PROGRAM P_PersistentDataSave
VAR
	fbSaveChanges :FB_Save;
	sFolderPath: STRING(255) := 'C:\Recipe_changes\';
END_VAR

IF P_persistent.bWritePersistent THEN
	fbSaveChanges.sFilePath := CONCAT(sFolderPath, 'Recipe_change');
    fbSaveChanges.sFilePath := CONCAT(fbSaveChanges.sFilePath, p_24h_C1_2.sCurrentDate);
    fbSaveChanges.sFilePath := CONCAT(fbSaveChanges.sFilePath, '.csv');
	fbSaveChanges();
END_IF

END_PROGRAM

(* stored: Version 1.1.0.1, ProductVersion 3.1.4026.13, FileIdentifier 561e912806da75a3470abee4b195e8b78ff5e6da, FileSignature 91b75a5166293d134c0b4d7ecb5ce9b6fdae071e385e36b36b597e2cd0a9c5db319be4bb0085fbdef6d3f87e57cd36932b6f82a5252ae615b6c7f43b9443b1043f2c0b209d572fa54bcda1dca1b0398354b0326b3359d55d822382cf1c3edfa60be165cb5de292d94b2cbdb23731b02ccfb9a12fa71c383b30162ebdaad2e779ab67d02c0a07b0d48d40d38076bb917bad770cd25abfd7a4e73f2d3cefd1385e6efad9fa0d90c2a3478c4bb024a861ae45c413af1536a2afe72560ca964263407b4bc7a9115b2b56d6a1af721a56582b8c7856729a774ae768ec496ed43b32a8741c9031995ab2080c8dbdbc07ce8d331f11b59eaa675c51d1a28f243c5f5167
   POU P_PersistentDataSave: Id {5f5e01b5-ade5-4ee8-97a0-229289adfb81}, SpecialFunc None *)
